// Mitsubishi GX Works2 project: auto_palletize_with_servo_dock   PLC: Q03UDV

PROGRAM MAIN
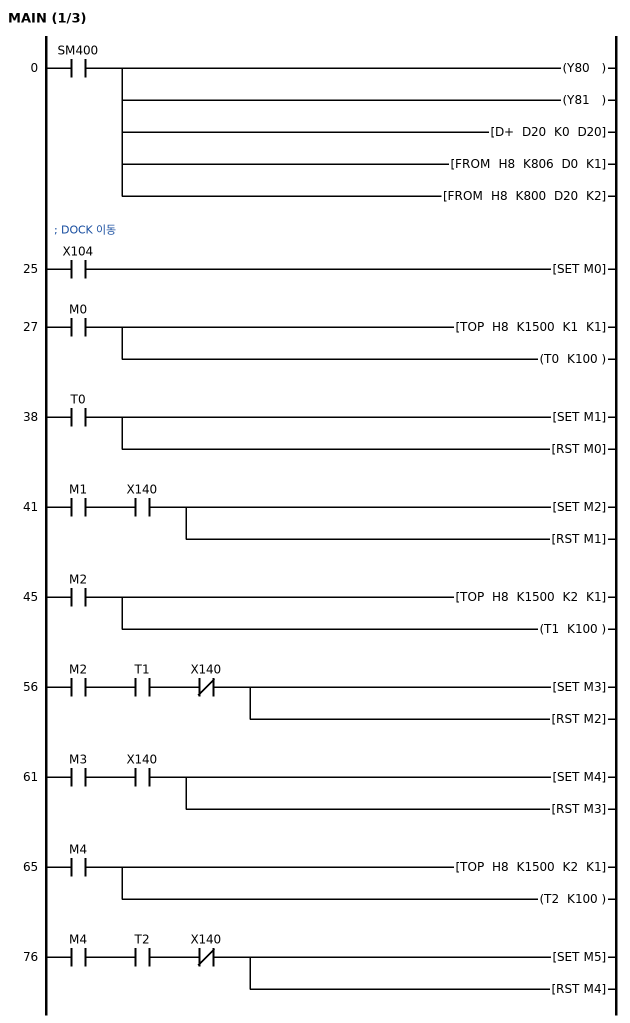
0     LD      SM400
      OUT     Y80
      OUT     Y81
      D+      D20 K0 D20
      FROM    H8 K806 D0 K1
      FROM    H8 K800 D20 K2
; DOCK 이동
25    LD      X104
      SET     M0
27    LD      M0
      TOP     H8 K1500 K1 K1
      OUT     T0 K100
38    LD      T0
      SET     M1
      RST     M0
41    LD      M1
      AND     X140
      SET     M2
      RST     M1
45    LD      M2
      TOP     H8 K1500 K2 K1
      OUT     T1 K100
56    LD      M2
      AND     T1
      ANI     X140
      SET     M3
      RST     M2
61    LD      M3
      AND     X140
      SET     M4
      RST     M3
65    LD      M4
      TOP     H8 K1500 K2 K1
      OUT     T2 K100
76    LD      M4
      AND     T2
      ANI     X140
      SET     M5
      RST     M4
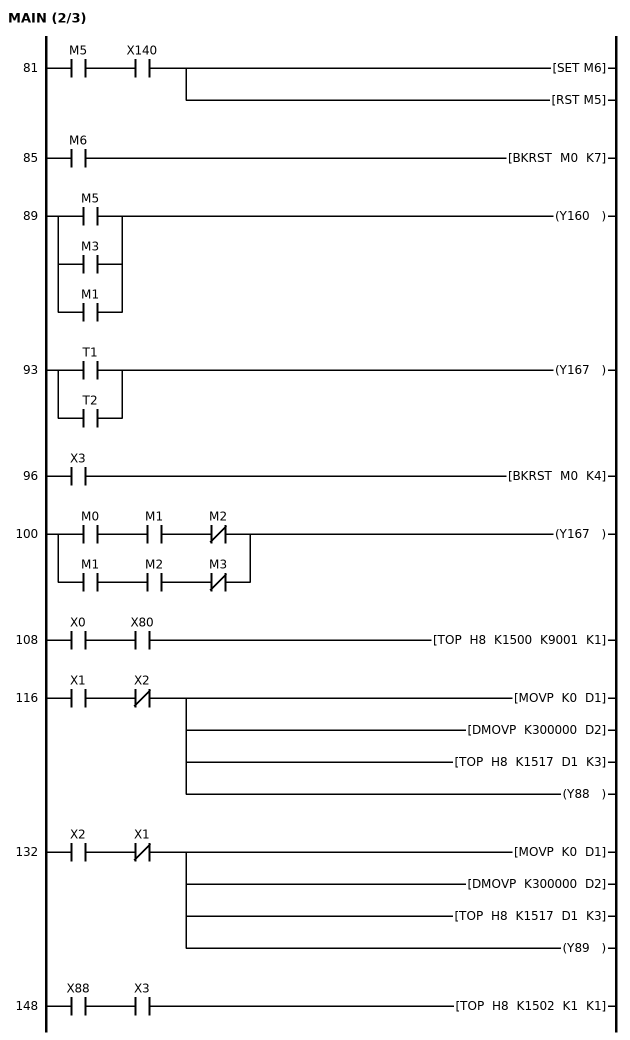
81    LD      M5
      AND     X140
      SET     M6
      RST     M5
85    LD      M6
      BKRST   M0 K7
89    LD      M5
      OR      M3
      OR      M1
      OUT     Y160
93    LD      T1
      OR      T2
      OUT     Y167
96    LD      X3
      BKRST   M0 K4
100   LD      M0
      AND     M1
      ANI     M2
      LD      M1
      AND     M2
      ANI     M3
      ORB
      OUT     Y167
108   LD      X0
      AND     X80
      TOP     H8 K1500 K9001 K1
116   LD      X1
      ANI     X2
      MOVP    K0 D1
      DMOVP   K300000 D2
      TOP     H8 K1517 D1 K3
      OUT     Y88
132   LD      X2
      ANI     X1
      MOVP    K0 D1
      DMOVP   K300000 D2
      TOP     H8 K1517 D1 K3
      OUT     Y89
148   LD      X88
      AND     X3
      TOP     H8 K1502 K1 K1
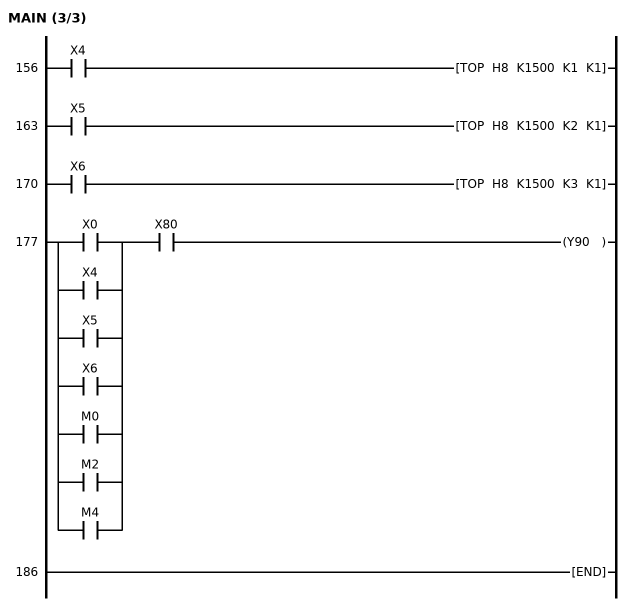
156   LD      X4
      TOP     H8 K1500 K1 K1
163   LD      X5
      TOP     H8 K1500 K2 K1
170   LD      X6
      TOP     H8 K1500 K3 K1
177   LD      X0
      OR      X4
      OR      X5
      OR      X6
      OR      M0
      OR      M2
      OR      M4
      AND     X80
      OUT     Y90
186   END
END_PROGRAM
